PROGRAM com_task
VAR
	try : BOOL := FALSE;
END_VAR

(* Zähler *)
Zaehler();

(* Wetterstation *)
Wetterstation();


try :=  TRUE;

END_PROGRAM

(* stored: Version 1.1.0.1, ProductVersion 3.1.4024.9
   POU com_task: Id {2a6820b0-4f66-4d85-a976-c6f73a5f0ae5}, SpecialFunc None *)
